// TwinCAT 3 PLC project PLC
// ProgramVersion: 3.1.4024.0
// libraries:
//   Tc2_Standard, * (Beckhoff Automation GmbH)
//   Tc2_System, * (Beckhoff Automation GmbH)
//   Tc2_Utilities, * (Beckhoff Automation GmbH)
//   Tc3_IotBase, * (Beckhoff Automation GmbH)
//   Tc3_JsonXml, * (Beckhoff Automation GmbH)
//   Tc3_Module, * (Beckhoff Automation GmbH)
//   Util, * (System)
// project tree:
//   / PlcTask.TcTTO
//   POUs/ FB_MQTT_Historize.TcPOU, FB_UnixTimestamp.TcPOU, FB_Values.TcPOU, MAIN.TcPOU
// real-time tasks:
//   TASK PlcTask: cycle T#10ms, priority 20, ADS port 350

CONFIGURATION PLC
    RESOURCE PLC ON TwinCAT3
        TASK PlcTask(INTERVAL := T#10ms, PRIORITY := 20);
        PROGRAM MAIN WITH PlcTask : MAIN;
    END_RESOURCE
END_CONFIGURATION

// ---- POUs/MAIN.TcPOU
PROGRAM MAIN
VAR
	

//runtime counter
	iCounter: INT;
	
//historize data
	fbMqttHistorize:FB_MQTT_Historize;
	
END_VAR

(*

-Test MQTT history values

*)

iCounter := iCounter +1;


fbMqttHistorize();

END_PROGRAM

// ---- POUs/FB_MQTT_Historize.TcPOU
FUNCTION_BLOCK FB_MQTT_Historize
VAR_INPUT
END_VAR
VAR_OUTPUT
END_VAR
VAR

//MQTT connection	
	fbMqttClient 					: FB_IotMqttClient;										//mqtt client
	bSetParameter 					: BOOL := TRUE;										//set parameter
	bConnect 						: BOOL := TRUE;										//connect to broker
	hrErrorOccurred 				: HRESULT;											//error ococured
	sTopicPubFast	 				: STRING(255) := 'historizeData/historizeFast';		//topic publich
	sTopicPubMiddle	 				: STRING(255) := 'historizeData/historizeMiddle';	//topic publich
	sTopicPubSlow	 				: STRING(255) := 'historizeData/historizeSlow';		//topic publich
	sPayloadPubFast					: STRING(1000);										//payload publish
	sPayloadPubMiddle				: STRING(1000);										//payload publish
	sPayloadPubSlow					: STRING(1000);										//payload publish
	fbMessageQueue 					: FB_IotMqttMessageQueue;							//message queue
	fbMessage 						: FB_IotMqttMessage;								//mqtt messaege
	{attribute 'TcEncoding':='UTF-8'}	
	sTopicRcv : STRING(255);															//topic received
	{attribute 'TcEncoding':='UTF-8'}
	sPayloadRcv : STRING(255);															//payload received
	
//json document
	fbJsonFast      					: FB_JsonSaxWriter;			//json sax write for payload
	fbJsonMiddle      					: FB_JsonSaxWriter;			//json sax write for payload
	fbJsonSlow  	   					: FB_JsonSaxWriter;			//json sax write for payload

//unix timestamp creation
	unixTime: FB_UnixTimestamp;									//create unit timestamp
    timestampSeconds: ULINT;									//unix timestamp second
    timestampMilliseconds: ULINT;								//unix timestamp milliseconds
	
//update timers	
	tonUpdateFast: TON;											//timer update data fast
	tonUpdateSlow: TON;											//timer update data slow
	tonUpdateMiddle: TON;
	
//value simulation	
	fbSimValues:FB_Values;										//simulate values

END_VAR

(*

-historize data with mqtt/telegraf/influxdb

*)


//simulate values
fbSimValues();

//generate unix time
unixTime(ulSeconds=> timestampSeconds, ulMilliseconds=>timestampMilliseconds );


//init connection parameter
IF bSetParameter THEN
	bSetParameter := FALSE;
	
	//broker settings for mosquitto w/o sec
	fbMqttClient.sHostName:= '192.168.1.50';
	fbMqttClient.nHostPort:= 1883;
	fbMqttClient.sClientId:= 'MqttHistorianPlcClient'; 

	fbMqttClient.ipMessageQueue := fbMessageQueue;
END_IF

//excute connect
fbMqttClient.Execute(bConnect);

//check error
IF fbMqttClient.bError THEN
	// add your error logging here
	hrErrorOccurred := fbMqttClient.hrErrorCode;
END_IF

//check queue messages
IF fbMessageQueue.nQueuedMessages > 0 THEN
	IF fbMessageQueue.Dequeue(fbMessage:=fbMessage) THEN
		fbMessage.GetTopic(pTopic:=ADR(sTopicRcv), nTopicSize:=SIZEOF(sTopicRcv) );
		fbMessage.GetPayload(pPayload:=ADR(sPayloadRcv), nPayloadSize:=SIZEOF(sPayloadRcv), bSetNullTermination:=FALSE);
	END_IF
END_IF

//cyclic update
tonUpdateFast(IN:=NOT tonUpdateFast.Q , PT:=T#250MS);
tonUpdateMiddle(IN:=NOT tonUpdateMIddle.Q , PT:=T#1S);
tonUpdateSlow(IN:=NOT tonUpdateSlow.Q , PT:=T#10S);


//publish fast values
IF fbMqttClient.bConnected  THEN
	
		//build JsonDoc
		BuildJsonDoc();	
		
		//send data fast
		IF tonUpdateFast.Q THEN
			//publish Values
			fbMqttClient.Publish(	sTopic:= sTopicPubFast, 
									pPayload:= ADR(sPayloadPubFast), nPayloadSize:= LEN2(ADR(sPayloadPubFast)), 
									eQoS:= TcIotMqttQos.AtMostOnceDelivery, bRetain:= FALSE, bQueue:= FALSE );
		END_IF
		
		//send data middle
		IF tonUpdateMiddle.Q THEN
			//publish Values
			fbMqttClient.Publish(	sTopic:= sTopicPubMiddle, 
									pPayload:= ADR(sPayloadPubMiddle), nPayloadSize:= LEN2(ADR(sPayloadPubMIddle)), 
									eQoS:= TcIotMqttQos.AtMostOnceDelivery, bRetain:= FALSE, bQueue:= FALSE );
		END_IF
				

		//send data slow
		IF tonUpdateSlow.Q THEN
			//publish Values
			fbMqttClient.Publish(	sTopic:= sTopicPubSlow, 
									pPayload:= ADR(sPayloadPubSlow), nPayloadSize:= LEN2(ADR(sPayloadPubSlow)), 
									eQoS:= TcIotMqttQos.AtMostOnceDelivery, bRetain:= FALSE, bQueue:= FALSE );
		END_IF
				
		//check pub erorrs						
		IF fbMqttClient.bError THEN
				// add your error logging here			
				hrErrorOccurred := fbMqttClient.hrErrorCode;
		END_IF
		
		
END_IF

METHOD BuildJsonDoc : BOOL
VAR_INPUT
END_VAR
(*

-generate JSON String

*)

		//generate fast json
		fbJsonFast.ResetDocument();
		fbJsonFast.SetMaxDecimalPlaces(2);	
		fbJsonFast.StartObject();
		fbJsonFast.AddKey('Timestamp');
		fbJsonFast.AddUlint(timestampMilliseconds);
		fbJsonFast.AddKeyLreal('Value01', fbSimValues.CosineSlow);
		fbJsonFast.AddKeyLreal('Value02', fbSimValues.sineSlow + 10);
		fbJsonFast.AddKeyLreal('Value03', fbSimValues.CosineSlow - 10);
		fbJsonFast.AddKeyLreal('Value04', fbSimValues.sineSlow + 20);
		fbJsonFast.AddKeyLreal('Value05', fbSimValues.CosineSlow - 20);
		fbJsonFast.AddKeyLreal('Value06', fbSimValues.sineSlow + 30);
		fbJsonFast.AddKeyLreal('Value07', fbSimValues.TriangleSlow);
		fbJsonFast.AddKeyLreal('Value08', fbSimValues.CosineSlow + 5);
		fbJsonFast.AddKeyLreal('Value09', fbSimValues.TriangleSlow + 3);
		fbJsonFast.AddKeyLreal('Value10', fbSimValues.CosineSlow + 6);
		fbJsonFast.EndObject();	
		fbJsonFast.CopyDocument(sPayloadPubFast, fbJsonFast.GetDocumentLength());
		
		
		
		//generate middle json
		fbJsonMIddle.ResetDocument();
		fbJsonMIddle.SetMaxDecimalPlaces(2);	
		fbJsonMIddle.StartObject();
		fbJsonMIddle.AddKey('Timestamp');
		fbJsonMIddle.AddUlint(timestampMilliseconds);
		fbJsonMIddle.AddKeyLreal('Value01', fbSimValues.CosineSlow);
		fbJsonMIddle.AddKeyLreal('Value02', fbSimValues.sineSlow + 10);
		fbJsonMIddle.AddKeyLreal('Value03', fbSimValues.CosineSlow - 10);
		fbJsonMIddle.AddKeyLreal('Value04', fbSimValues.sineSlow + 20);
		fbJsonMIddle.AddKeyLreal('Value05', fbSimValues.CosineSlow - 20);
		fbJsonMIddle.AddKeyLreal('Value06', fbSimValues.sineSlow + 30);
		fbJsonMIddle.AddKeyLreal('Value07', fbSimValues.TriangleSlow);
		fbJsonMIddle.AddKeyLreal('Value08', fbSimValues.CosineSlow + 5);
		fbJsonMIddle.AddKeyLreal('Value09', fbSimValues.TriangleSlow + 3);
		fbJsonMIddle.AddKeyLreal('Value10', fbSimValues.CosineSlow + 6);
		fbJsonMIddle.EndObject();	
		fbJsonMIddle.CopyDocument(sPayloadPubMIddle, fbJsonMIddle.GetDocumentLength());
		
		
		//generate Slow json
		fbJsonSlow.ResetDocument();
		fbJsonSlow.SetMaxDecimalPlaces(2);	
		fbJsonSlow.StartObject();
		fbJsonSlow.AddKey('Timestamp');
		fbJsonSlow.AddUlint(timestampMilliseconds);
		fbJsonSlow.AddKeyLreal('Value01', fbSimValues.CosineSlow);
		fbJsonSlow.AddKeyLreal('Value02', fbSimValues.sineSlow + 10);
		fbJsonSlow.AddKeyLreal('Value03', fbSimValues.CosineSlow - 10);
		fbJsonSlow.AddKeyLreal('Value04', fbSimValues.sineSlow + 20);
		fbJsonSlow.AddKeyLreal('Value05', fbSimValues.CosineSlow - 20);
		fbJsonSlow.AddKeyLreal('Value06', fbSimValues.sineSlow + 30);
		fbJsonSlow.AddKeyLreal('Value07', fbSimValues.TriangleSlow);
		fbJsonSlow.AddKeyLreal('Value08', fbSimValues.CosineSlow + 5);
		fbJsonSlow.AddKeyLreal('Value09', fbSimValues.TriangleSlow + 3);
		fbJsonSlow.AddKeyLreal('Value10', fbSimValues.CosineSlow + 6);
		fbJsonSlow.EndObject();	
		fbJsonSlow.CopyDocument(sPayloadPubSlow, fbJsonSlow.GetDocumentLength());
END_METHOD

END_FUNCTION_BLOCK

// ---- POUs/FB_UnixTimestamp.TcPOU
FUNCTION_BLOCK FB_UnixTimestamp
VAR_INPUT
END_VAR
VAR_OUTPUT
	ulSeconds: ULINT;		//Seconds
    ulMilliseconds: ULINT;	///Milliseconds
END_VAR
VAR
	fbLocalSystemTime : FB_LocalSystemTime;
    fbGetTimeZoneInformation : FB_GetTimeZoneInformation;
    stTimeZoneInformation : ST_TimeZoneInformation;
    fbTzSpecificLocalTimeToFileTime : FB_TzSpecificLocalTimeToFileTime;
    tFileTime: T_FILETIME;
    onZerothSecondLastCycle : BOOL;
END_VAR

(*

-convert to unix timestamp
https://stackoverflow.com/questions/41773732/how-do-i-get-the-unix-timestamp-in-twincat3

*)

// Get local system time
fbLocalSystemTime(bEnable:=TRUE, dwCycle:=1);

// On the zeroth second of each minutesync timezone information
IF (stTimeZoneInformation.standardName = '' OR (fbLocalSystemTime.systemTime.wSecond = 0 AND NOT onZerothSecondLastCycle)) THEN
    fbGetTimeZoneInformation(sNetID := '', bExecute := TRUE, tzInfo => stTimeZoneInformation);
END_IF;

//convert to unix timestamp
fbTzSpecificLocalTimeToFileTime(in := Tc2_Utilities.SYSTEMTIME_TO_FILETIME(fbLocalSystemTime.systemTime), tzInfo := stTimeZoneInformation, out => tFileTime);
ulSeconds := (SHL(DWORD_TO_ULINT(tFileTime.dwHighDateTime), 32) + DWORD_TO_ULINT(tFileTime.dwLowDateTime)) / 10000000 - 11644473600;
ulMilliseconds := (SHL(DWORD_TO_ULINT(tFileTime.dwHighDateTime), 32) + DWORD_TO_ULINT(tFileTime.dwLowDateTime)) / 10000 - 11644473600000;

onZerothSecondLastCycle := fbLocalSystemTime.systemTime.wSecond = 0;

END_FUNCTION_BLOCK

// ---- POUs/FB_Values.TcPOU
FUNCTION_BLOCK FB_Values
VAR_INPUT
END_VAR
VAR_OUTPUT
END_VAR
VAR

//Function Blocks	
	fbSineFast:GEN;
	fbCosineFast:GEN;
	fbTriangleFast:GEN;
	fbSineSlow:GEN;
	fbCosineSlow:GEN;
	fbTriangleSlow:GEN;
	
//FB Outputs
	iSineFast: INT;
	iCosineFast: INT;
	iTriangleFast: INT;
	iSineSlow: INT;
	iCosineSlow: INT;
	iTriangleSlow: INT;
	
END_VAR

(*
-signal generator

*)

//sine fast
fbSineFast(
	MODE:=SINE , 
	BASE:=TRUE , 
	PERIOD:=T#500MS , 
	CYCLES:= , 
	AMPLITUDE:=100 , 
	RESET:= , 
	OUT=>iSineFast );
	
//cosine
fbCoSineFast(
	MODE:=COSINE , 
	BASE:=TRUE , 
	PERIOD:=T#600MS , 
	CYCLES:= , 
	AMPLITUDE:=100 , 
	RESET:= , 
	OUT=>iCosineFast );

//triangular
fbTriangleFast(
	MODE:=TRIANGLE , 
	BASE:=TRUE , 
	PERIOD:=T#700MS , 
	CYCLES:= , 
	AMPLITUDE:=200 , 
	RESET:= , 
	OUT=>iTriangleFast );


//sine
fbSineSlow(
	MODE:=SINE , 
	BASE:=TRUE , 
	PERIOD:=T#5S , 
	CYCLES:= , 
	AMPLITUDE:=100 , 
	RESET:= , 
	OUT=>iSineSlow );
	
//cosine
fbCoSineSlow(
	MODE:=COSINE , 
	BASE:=TRUE , 
	PERIOD:=T#6S , 
	CYCLES:= , 
	AMPLITUDE:=100 , 
	RESET:= , 
	OUT=>iCosineSlow );

//triangular
fbTriangleSlow(
	MODE:=TRIANGLE , 
	BASE:=TRUE , 
	PERIOD:=T#7S , 
	CYCLES:= , 
	AMPLITUDE:=200 , 
	RESET:= , 
	OUT=>iTriangleSlow );

PROPERTY CosineFast : REAL
GET
CosineFast:=TO_REAL(iCosineFast);
END_GET
END_PROPERTY

PROPERTY CosineSlow : REAL
GET
CosineSlow:=TO_REAL(iCosineSlow);
END_GET
END_PROPERTY

PROPERTY SineFast : REAL
GET
SineFast:=TO_REAL(iSineFast);
END_GET
END_PROPERTY

PROPERTY SineSlow : REAL
GET
SineSlow:=TO_REAL(iSineFast);
END_GET
END_PROPERTY

PROPERTY TriangleFast : REAL
GET
TriangleFast:=TO_REAL(iTriangleFast);
END_GET
END_PROPERTY

PROPERTY TriangleSlow : REAL
GET
TriangleSlow:=TO_REAL(iTriangleSlow);
END_GET
END_PROPERTY

END_FUNCTION_BLOCK
